# B&R Automation Studio project Panel
Automation Studio 3.0.90.22 SP04


## Logical view

Binary libraries used (declarations not repeated): operator, runtime, astime, AsIecCon, asstring, AsARCfg, FileIO, AsTCP, visapi

### Global.typ - Global data types
```iecst
(********************************************************************
 * COPYRIGHT --
 ********************************************************************
 * File: Global.typ
 * Author: florian
 * Created: November 16, 2012
 ********************************************************************
 * Global data types of project CANOpenMaster
 ********************************************************************)

TYPE
	LibVisapi5_ST_state_type : 	STRUCT  (*State variables of VISAPI commands*)
		va_srelease : UINT; (*State variable of command VA_Srelease*)
		va_saccess : UINT; (*State variable of command VA_Saccess*)
		va_loadbitmap : UINT; (*State variable of command VA_LoadBitmap*)
		va_blitbitmap : UINT; (*State variable of command VA_BlitBitmap*)
		va_freebitmap : UINT; (*State variable of command VA_FreeBitmap*)
		va_attach : UINT; (*State variable of command VA_Attach*)
		va_detach : UINT; (*State variable of command VA_Detach*)
		va_redraw : UINT; (*State variable of command VA_Redraw*)
		bmpcase : UINT;
	END_STRUCT;
END_TYPE
```

### Global.var - Global variables
```iecst
(********************************************************************
 * COPYRIGHT --
 ********************************************************************
 * File: Global.var
 * Author: florian
 * Created: November 16, 2012
 ********************************************************************
 * Global variables of project CANOpenMaster
 ********************************************************************)
VAR
	GetPage : INT;
	SetPage : INT;
	Strings : ARRAY[0..99] OF STRING[42];
	Action : UINT;
	Selection : UINT;
	Search : STRING[80];
	Limit : UINT;
	OFF : USINT := 0;
	state : LibVisapi5_ST_state_type; (*State variables of VISAPI commands*)
	Edit : UINT;
	VC_HANDLE : UDINT;
	ready : DINT;
	blnState : UDINT;
END_VAR
```


### Program Logical/FTP/FTP (IEC) - Network file system configuration

#### FTP.st - Implementation code
```iecst
(********************************************************************
 * COPYRIGHT -- Bernecker + Rainer
 ********************************************************************
 * Program: NwFileSystem
 * File: NwFileSystem.st
 * Author: Bernecker + Rainer
 * Created: April 21, 2009
 ********************************************************************
 * Implementation of program NwFileSystem
 ********************************************************************)

PROGRAM _INIT

	(* Init values *)
	strcpy(ADR(Network.Data.Device), ADR('IF2'));  (* X20 CPU Ethernet device *)

END_PROGRAM

PROGRAM _CYCLIC

	CASE Network.Data.Step OF

		0:	IF Network.Command.bCfgSetFTPServer = 1 THEN
				Network.Data.Step := 10;
			ELSIF Network.Command.bCfgGetCIFSDefaultuser = 1 THEN
				Network.Data.Step := 20;
			ELSIF Network.Command.bCfgSetCIFSDefaultuser = 1 THEN
				Network.Data.Step := 30;
			ELSIF Network.Command.bCfgGetCIFSDomain = 1 THEN
				Network.Data.Step := 40;
			ELSIF Network.Command.bCfgSetCIFSDomain = 1 THEN
				Network.Data.Step := 50;
			END_IF

		10:  (* Enable/disable the FTP server *)
			Network.Functionblocks.CfgSetFTPServer_0.enable := 1;  (* Enable the function block *)
			Network.Functionblocks.CfgSetFTPServer_0.Option := cfgOPTION_ENABLE;  (* Enable FTP server *)

			Network.Functionblocks.CfgSetFTPServer_0;  (* Function Call *)

			IF Network.Functionblocks.CfgSetFTPServer_0.status = 0 THEN  (* CfgSetFTPServer successfull *)
				Network.Command.bCfgSetFTPServer := 0;
				Network.Data.Step := 0;
			ELSIF Network.Functionblocks.CfgSetFTPServer_0.status = ERR_FUB_BUSY THEN  (* CfgSetHostName not finished -> redo *)
				(* Busy *)
			ELSE  (* Goto Error Step *)
				Network.Data.Step := 255;
			END_IF

		20:  (* Read the CIFS default user settings *)
			Network.Functionblocks.CfgGetCIFSDefaultuser_0.enable := 1;  (* Enable the function block *)
			Network.Functionblocks.CfgGetCIFSDefaultuser_0.pDefaultuser := ADR(Network.Data.DefaultUser);  (* Address of the DefaultUser string *)
			Network.Functionblocks.CfgGetCIFSDefaultuser_0.lenUser := SIZEOF(Network.Data.DefaultUser);  (* Length of the DefaultUser string *)
			Network.Functionblocks.CfgGetCIFSDefaultuser_0.pDefaultpassword := ADR(Network.Data.DefaultPassword);  (* Address of the DefaultPassword string *)
			Network.Functionblocks.CfgGetCIFSDefaultuser_0.lenPassword := SIZEOF(Network.Data.DefaultPassword);  (* Length of the DefaultPassword string *)

			Network.Functionblocks.CfgGetCIFSDefaultuser_0;  (* Function Call *)

			IF Network.Functionblocks.CfgGetCIFSDefaultuser_0.status = 0 THEN  (* CfgGetCIFSDefaultuser successfull *)
				Network.Command.bCfgGetCIFSDefaultuser := 0;
				Network.Data.Step := 0;
			ELSIF Network.Functionblocks.CfgGetCIFSDefaultuser_0.status = ERR_FUB_BUSY THEN  (* CfgGetCIFSDefaultuser not finished -> redo *)
				(* Busy *)
			ELSE  (* Goto Error Step *)
				Network.Data.Step := 255;
			END_IF

		30:  (* Modify the settings of the CIFS default user *)
			Network.Functionblocks.CfgSetCIFSDefaultuser_0.enable := 1;  (* Enable the function block *)
			Network.Functionblocks.CfgSetCIFSDefaultuser_0.pDefaultuser := ADR(Network.Data.DefaultUser);  (* Address of the DefaultUser string *)
			Network.Functionblocks.CfgSetCIFSDefaultuser_0.pDefaultpassword := ADR(Network.Data.DefaultPassword);  (* Address of the DefaultPassword string *)
			Network.Functionblocks.CfgSetCIFSDefaultuser_0.Option := cfgOPTION_NON_VOLATILE;  (*  Temporarily set the parameter *)

			Network.Functionblocks.CfgSetCIFSDefaultuser_0;  (* Function Call *)

			IF Network.Functionblocks.CfgSetCIFSDefaultuser_0.status = 0 THEN  (* CfgSetCIFSDefaultuser successfull *)
				Network.Command.bCfgSetCIFSDefaultuser := 0;
				Network.Data.Step := 0;
			ELSIF Network.Functionblocks.CfgSetCIFSDefaultuser_0.status = ERR_FUB_BUSY THEN  (* CfgSetCIFSDefaultuser not finished -> redo *)
				(* Busy *)
			ELSE  (* Goto Error Step *)
				Network.Data.Step := 255;
			END_IF

		40:  (* Read the domain configurations for CIFS *)
			Network.Functionblocks.CfgGetCIFSDomain_0.enable := 1;  (* Enable the function block *)
			Network.Functionblocks.CfgGetCIFSDomain_0.pDomain := ADR(Network.Data.Domain);  (* Address of the Domain string *)
	  		Network.Functionblocks.CfgGetCIFSDomain_0.Len := SIZEOF(Network.Data.Domain);  (* Length of the Domain string *)

			Network.Functionblocks.CfgGetCIFSDomain_0;  (* Function Call *)

			IF Network.Functionblocks.CfgGetCIFSDomain_0.status = 0 THEN  (* CfgGetCIFSDomain successfull *)
				Network.Data.Workgroup := Network.Functionblocks.CfgGetCIFSDomain_0.isWorkgroup;
				Network.Command.bCfgGetCIFSDomain := 0;
				Network.Data.Step := 0;
			ELSIF Network.Functionblocks.CfgGetCIFSDomain_0.status = ERR_FUB_BUSY THEN  (* CfgGetCIFSDomain not finished -> redo *)
				(* Busy *)
			ELSE  (* Goto Error Step *)
				Network.Data.Step := 255;
			END_IF

		50:  (* Edit the domain configurations for CIFS *)
			Network.Functionblocks.CfgSetCIFSDomain_0.enable := 1;  (* Enable the function block *)
			Network.Functionblocks.CfgSetCIFSDomain_0.pDomain := ADR(Network.Data.Domain);  (* Address of the Domain string *)
			Network.Functionblocks.CfgSetCIFSDomain_0.isWorkgroup := Network.Data.Workgroup;
			Network.Functionblocks.CfgSetCIFSDomain_0.Option := cfgOPTION_NON_VOLATILE;  (*  Temporarily set the parameter *)

			Network.Functionblocks.CfgSetCIFSDomain_0;  (* Function Call *)

			IF Network.Functionblocks.CfgSetCIFSDomain_0.status = 0 THEN  (* CfgSetCIFSDomain successfull *)
				Network.Command.bCfgSetCIFSDomain := 0;
				Network.Data.Step := 0;
			ELSIF Network.Functionblocks.CfgSetCIFSDomain_0.status = ERR_FUB_BUSY THEN  (* CfgSetCIFSDomain not finished -> redo *)
				(* Busy *)
			ELSE  (* Goto Error Step *)
				Network.Data.Step := 255;
			END_IF

		255:  (*Error handling*)

	END_CASE

END_PROGRAM
```

#### FTP.typ - Local data types
```iecst
(********************************************************************
 * COPYRIGHT -- Bernecker + Rainer
 ********************************************************************
 * Program: NwFileSystem
 * File: NwFileSystem.typ
 * Author: Bernecker + Rainer
 * Created: April 21, 2009
 ********************************************************************
 * Local data types of program NwFileSystem
 ********************************************************************)

TYPE
	Network_typ : 	STRUCT
		Command : Network_Command_typ; (*Structure Command (contains all command elements)*)
		Data : Network_Data_typ; (*Structure Data (contains all data informations)*)
		Functionblocks : Network_Functionblocks_typ; (*Structure Functionblocks (contains all FuBs)*)
	END_STRUCT;
	Network_Command_typ : 	STRUCT
		bCfgSetFTPServer : BOOL; (*Command: Start the FTP server*)
		bCfgGetCIFSDefaultuser : BOOL; (*Command: Get CIFS default user settings*)
		bCfgSetCIFSDefaultuser : BOOL; (*Command: Set CIFS default user settings*)
		bCfgGetCIFSDomain : BOOL; (*Command: Get CIFS domain configuration*)
		bCfgSetCIFSDomain : BOOL; (*Command: Set CIFS domain configuration*)
	END_STRUCT;
	Network_Data_typ : 	STRUCT
		DefaultUser : STRING[80]; (*Data variable for CfgGetCIFSDefaultuser() and CfgSetCIFSDefaultuser()*)
		DefaultPassword : STRING[80]; (*Data variable for CfgGetCIFSDefaultuser() and CfgSetCIFSDefaultuser()*)
		Domain : STRING[80]; (*Data variable for CfgGetCIFSDomain() and CfgSetCIFSDomain()*)
		Workgroup : USINT; (*Data variable for CfgGetCIFSDomain() and CfgSetCIFSDomain()*)
		Device : STRING[80]; (*Device string (contains the device path)*)
		Step : USINT; (*Step variable*)
	END_STRUCT;
	Network_Functionblocks_typ : 	STRUCT
		CfgSetFTPServer_0 : CfgSetFTPServer; (*Functionblock CfgSetFTPServer()*)
		CfgGetCIFSDefaultuser_0 : CfgGetCIFSDefaultuser; (*Functionblock CfgGetCIFSDefaultuser()*)
		CfgSetCIFSDefaultuser_0 : CfgSetCIFSDefaultuser; (*Functionblock CfgSetCIFSDefaultuser()*)
		CfgGetCIFSDomain_0 : CfgGetCIFSDomain; (*Functionblock CfgGetCIFSDomain()*)
		CfgSetCIFSDomain_0 : CfgSetCIFSDomain; (*Functionblock CfgSetCIFSDomain()*)
	END_STRUCT;
END_TYPE
```

#### FTP.var - Local variables
```iecst
(********************************************************************
 * COPYRIGHT -- Bernecker + Rainer
 ********************************************************************
 * Program: NwFileSystem
 * File: NwFileSystem.var
 * Author: Bernecker + Rainer
 * Created: April 21, 2009
 ********************************************************************
 * Local variables of program NwFileSystem
 ********************************************************************)
VAR
	Network : Network_typ; (*Global structure*)
END_VAR
```

### Program Logical/handler (ANSIC) - A new program

#### handlerCyclic.c - Cyclic code
```c
/********************************************************************
 * COPYRIGHT --
 ********************************************************************
 * Program: handler
 * File: handlerCyclic.c
 * Author: florian
 * Created: January 06, 2013
 ********************************************************************
 * Implementation of program handler
 ********************************************************************/

#include <bur/plctypes.h>

#ifdef _DEFAULT_INCLUDES
	#include <AsDefault.h>
#endif

/****h* Panel/Panelhandler
* NAME
* 	Panelhandler
* FUNCTION
* 	This module contains the slave for the panel.
*
*****/

void _INIT handler(void){
	OFF=0;
	ready=0;
	VC_HANDLE=0;
	blnState=0;
}

/****f* Panel/load_image
* FUNCTION
* 	Function loads image from file and display it on screen.
*	Disabled by now because B&R uses a unusual image format
* SOURCE
*/
void load_image(){
	static int handle;
	if(handle == 0){
		handle = VA_Setup(1 , 'Visu'); //Get visualization handle
	} else {
		state.va_saccess = VA_Saccess(1,handle); //Get access to visualization *)
		if(state.va_saccess == 0){ // Check if access is OK *)
			switch(state.bmpcase){
				case 0:
					state.va_loadbitmap = VA_LoadBitmap(1, handle, "IMG", "0.png", &pBitmap);	// Load picture into memory
					if(state.va_loadbitmap == 0){
						//						state.va_redraw = VA_Redraw(1, handle); //Clean page befor drawing a new picture
						state.bmpcase++;
					}
					break;
				case 1:
					state.va_blitbitmap = VA_BlitBitmap(1, handle, pBitmap, 0, 0, 0, 0, 0, 0, 0);//Show picture at specific coordinates
					if(state.va_blitbitmap == 0)state.bmpcase++;
					break;
				case 2:
					state.va_freebitmap = VA_FreeBitmap(1, handle, &pBitmap); //Delete picture from memory
					if(state.va_freebitmap == 0){
					state.bmpcase++;
					}
				case 3:
					state.va_srelease = VA_Srelease(1, handle);
					state.bmpcase++;
					break;
			}
		}
	}
}
/*****/

/****f* Panel/handlerCyclic
* FUNCTION
*	This function is responsible for the page managment.
* SOURCE
*/
void _CYCLIC handlerCyclic(void)
{
	int i;

	SetPage=SetPage;
	GetPage=GetPage;
	Limit=Limit;
	Selection=Selection;

	for(i=0;i<100;i++){
		Search[i]=Search[i];
	}

	if(Action!=0){
		Edit=1;
		SetPage=0;
		Limit=0;
	}

	for(i=0;i<42;i++){
		Strings[i][0]=Strings[i][0];
	}

	if(GetPage==1){
		strcpy(Strings[0], "...Loading...");
		Strings[1][0]=0;
	}

	if(GetPage==3){
//		load_image();
	} else {
		state.bmpcase=0;
	}

	if(OFF!=0){
		Action=123;

		if (!ready)
		{
			VC_HANDLE = VA_Setup(1 , "Visu");
			if (VC_HANDLE)
				ready = 1;
		}
		if (ready)
		{
			if (!VA_Saccess(1,VC_HANDLE))
			{
				VA_SetBacklight(1,VC_HANDLE,blnState);
				VA_Srelease(1,VC_HANDLE);
			}
		}

	}

}
/*****/
```

#### handler.var - Local variables
```iecst
(********************************************************************
 * COPYRIGHT --
 ********************************************************************
 * Program: handler
 * File: handler.var
 * Author: florian
 * Created: January 06, 2013
 ********************************************************************
 * Local variables of program handler
 ********************************************************************)
VAR
	pBitmap : REFERENCE TO sVCBitmap;
END_VAR
```

- Visualisation Logical/Visu (not shown)
